FUNCTION_BLOCK Datatypes IMPLEMENTS I_Datatypes
VAR
	datatypes : Dictionary;
END_VAR

METHOD PUBLIC InsertByName
VAR_INPUT
	Name : T_MAXSTRING;
	Datatype : I_Datatype;
END_VAR
datatypes.AddOrUpdate(Name,Datatype);
END_METHOD

METHOD PUBLIC TryGetByName : BOOL
VAR_INPUT
	Name : T_MAXSTRING;
	Destination : REFERENCE TO I_Datatype;
END_VAR
TryGetByName := datatypes.TryGetValue(Name, Destination);
END_METHOD

END_FUNCTION_BLOCK

(* stored: Version 1.1.0.1, ProductVersion 3.1.4024.12
   POU Datatypes: Id {695b6b4a-c949-0743-1d47-4a41f3736c15}, SpecialFunc None
   Method InsertByName: Id {66c90401-a850-06d1-0c36-79dbafbbe7b4}
   Method TryGetByName: Id {0e472e8b-43d1-041b-35b0-54c91730f712} *)
